// TIA Portal V20 export
TYPE "UDT_Flowmeter_Status"
   STRUCT
      ISt_Flow_Aktuell : Real;
      Flow_smoothe_Value : Real;
      Ist_Temp_Aktuell : Real;
      Temp_smoothe_Value : Real;
      VISU_FARBE_Flow : Int;
      VISU_FARBE_Temp : Int;
      MESS_DB_STOE : Bool;
      Bit10 : Bool;
      Bit11 : Bool;
      Bit12 : Bool;
      Bit13 : Bool;
      Bit14 : Bool;
      Bit15 : Bool;
      Bit2_0 : Bool;
      Bit2_1 : Bool;
      Bit2_2 : Bool;
      Bit2_3 : Bool;
      Bit2_4 : Bool;
      Bit2_5 : Bool;
      Bit2_6 : Bool;
      Bit2_7 : Bool;
      Bit3_0 : Bool;
      Bit3_1 : Bool;
      Bit3_2 : Bool;
      Bit3_3 : Bool;
      Bit3_4 : Bool;
      Bit3_5 : Bool;
      Bit3_6 : Bool;
      Bit3_7 : Bool;
   END_STRUCT;
END_TYPE
